// TIA Portal project "topgun_plc" (V16)

(* hardware
DEVICE "S7-1200 station_1"  S7-1200 Station
   slot 0: "Rack_0"  S7-1200 Rack  Rack  V1.0
   slot 1: "PLC_CU"  CPU 1214C DC/DC/DC  6ES7 214-1AG40-0XB0  V4.4
   slot 2: "DI 16/DQ 16x24VDC_1"  6ES7 223-1BL32-0XB0  V2.0
   slot 3: "CB 1241 (RS485)"  CB 1241 (RS485)  6ES7 241-1CH30-1XB0  V1.0
DEVICE "S7-1200 station_2"  S7-1200 Station
   slot 0: "Rack_0"  S7-1200 Rack  Rack  V1.0
   slot 1: "PLC_CAM"  CPU 1214C DC/DC/DC  6ES7 214-1AG40-0XB0  V4.4
*)

// ===== PLC "PLC_CU"  CPU 1214C DC/DC/DC =====

VAR_GLOBAL   // PLC tag table "Default tag table"
   "System_Byte" AT %MB1 : Byte;
   "FirstScan" AT %M1.0 : Bool;
   "DiagStatusUpdate" AT %M1.1 : Bool;
   "AlwaysTRUE" AT %M1.2 : Bool;
   "AlwaysFALSE" AT %M1.3 : Bool;
   "Clock_Byte" AT %MB0 : Byte;
   "Clock_10Hz" AT %M0.0 : Bool;
   "Clock_5Hz" AT %M0.1 : Bool;
   "Clock_2.5Hz" AT %M0.2 : Bool;
   "Clock_2Hz" AT %M0.3 : Bool;
   "Clock_1.25Hz" AT %M0.4 : Bool;
   "Clock_1Hz" AT %M0.5 : Bool;
   "Clock_0.625Hz" AT %M0.6 : Bool;
   "Clock_0.5Hz" AT %M0.7 : Bool;
   "Tag_1" AT %I0.0 : Bool;
   "Tag_2" AT %I0.1 : Bool;
   "Tag_3" AT %I0.2 : Bool;
   "Tag_4" AT %I0.3 : Bool;
   "Tag_5" AT %I2.2 : Bool;
   "Tag_6" AT %I2.3 : Bool;
   "Tag_7" AT %I2.6 : Bool;
   "Tag_8" AT %I2.7 : Bool;
   "Tag_9" AT %ID1000 : DWord;
   "Tag_10" AT %ID1004 : DWord;
   "Tag_11" AT %ID1002 : DWord;
   "Tag_12" AT %ID1006 : DWord;
   "Tag_13" AT %M100.0 : Bool;
   "Tag_14" AT %M100.1 : Bool;
END_VAR

DATA_BLOCK "MB_CONFIG"   // DB2
{ S7_Optimized_Access := 'TRUE' }
VERSION : 0.1
   VAR
      MB_stat : Word;
      MB1_stat : Word;
      MB : TCON_IP_v4;
      MB1 : TCON_IP_v4;
   END_VAR
BEGIN
   MB.RemoteAddress.ADDR[1] := 16#C0;
   MB.RemoteAddress.ADDR[2] := 16#A8;
   MB.RemoteAddress.ADDR[4] := 16#49;
   MB.LocalPort := 502;
   MB1.RemoteAddress.ADDR[1] := 16#C0;
   MB1.RemoteAddress.ADDR[2] := 16#A8;
   MB1.RemoteAddress.ADDR[4] := 16#47;
   MB1.LocalPort := 503;
   MB.InterfaceId := 64;
   MB.ID := 2;
   MB1.InterfaceId := 64;
   MB1.ID := 3;
END_DATA_BLOCK

DATA_BLOCK "MB_DATA"   // DB3
{ S7_Optimized_Access := 'FALSE' }
VERSION : 0.1
   VAR
      DATA : Array[0..64] of Int;
   END_VAR
BEGIN
   DATA[4] := 6;
END_DATA_BLOCK

DATA_BLOCK "Retain_mem"   // DB7
{ S7_Optimized_Access := 'TRUE' }
VERSION : 0.1
   VAR
      Value_HSC1_Save : DWord;
   END_VAR
   VAR RETAIN
      Value_HSC1_Load : DWord;
   END_VAR
   VAR
      Value_HSC2_Save : DWord;
   END_VAR
   VAR RETAIN
      Value_HSC2_Load : DWord;
   END_VAR
   VAR
      Value_Angle1 : Real;
      Value_Angle2 : Real;
      temp1 : Real;
      temp2 : Real;
   END_VAR
BEGIN
END_DATA_BLOCK

ORGANIZATION_BLOCK "Main"   // OB1, LAD, ProgramCycle
TITLE = "Main Program Sweep (Cycle)"
{ S7_Optimized_Access := 'TRUE' }
VERSION : 0.1
   VAR_INPUT
      Initial_Call : Bool;   // Initial call of this OB
      Remanence : Bool;   // =True, if remanent data are available
   END_VAR
BEGIN

REGION Network 1
   // modbus 485
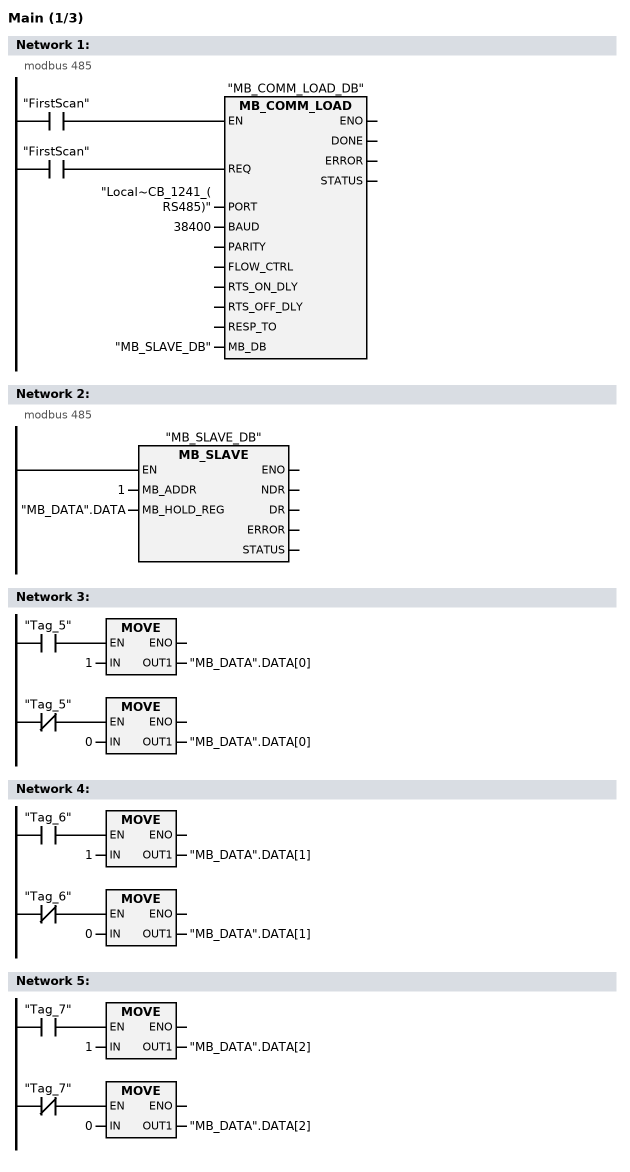
   IF "FirstScan" THEN
       "MB_COMM_LOAD_DB"(REQ := "FirstScan", PORT := "Local~CB_1241_(RS485)", BAUD := 38400, MB_DB := "MB_SLAVE_DB");   // MB_COMM_LOAD
   END_IF;
END_REGION

REGION Network 2
   // modbus 485
   "MB_SLAVE_DB"(MB_ADDR := 1, MB_HOLD_REG := "MB_DATA".DATA);   // MB_SLAVE
END_REGION

REGION Network 3
   RUNG wire#powerrail
      Contact( "Tag_5" )
      Move(in := 1, out1 => "MB_DATA".DATA[0])
   END_RUNG
   RUNG wire#powerrail
      I_Contact( "Tag_5" )
      Move(in := 0, out1 => "MB_DATA".DATA[0])
   END_RUNG
   // the same network as SCL:
   IF "Tag_5" THEN "MB_DATA".DATA[0] := 1; END_IF;
   IF NOT "Tag_5" THEN "MB_DATA".DATA[0] := 0; END_IF;
END_REGION

REGION Network 4
   RUNG wire#powerrail
      Contact( "Tag_6" )
      Move(in := 1, out1 => "MB_DATA".DATA[1])
   END_RUNG
   RUNG wire#powerrail
      I_Contact( "Tag_6" )
      Move(in := 0, out1 => "MB_DATA".DATA[1])
   END_RUNG
   // the same network as SCL:
   IF "Tag_6" THEN "MB_DATA".DATA[1] := 1; END_IF;
   IF NOT "Tag_6" THEN "MB_DATA".DATA[1] := 0; END_IF;
END_REGION

REGION Network 5
   RUNG wire#powerrail
      Contact( "Tag_7" )
      Move(in := 1, out1 => "MB_DATA".DATA[2])
   END_RUNG
   RUNG wire#powerrail
      I_Contact( "Tag_7" )
      Move(in := 0, out1 => "MB_DATA".DATA[2])
   END_RUNG
   // the same network as SCL:
   IF "Tag_7" THEN "MB_DATA".DATA[2] := 1; END_IF;
   IF NOT "Tag_7" THEN "MB_DATA".DATA[2] := 0; END_IF;
END_REGION

REGION Network 6
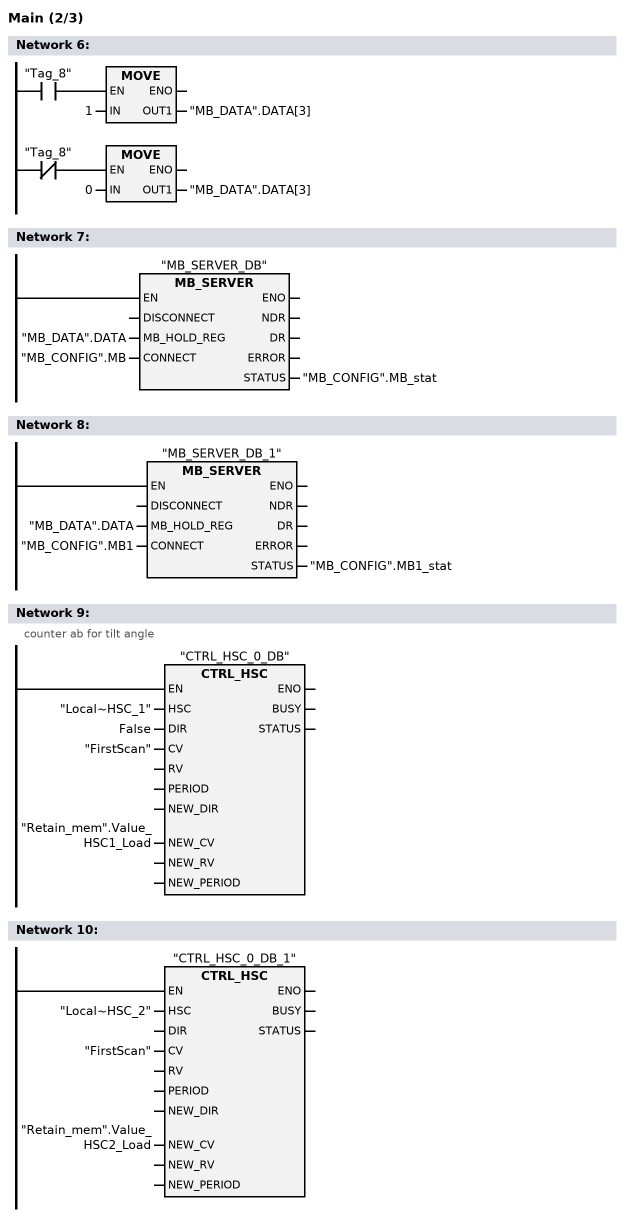
   RUNG wire#powerrail
      Contact( "Tag_8" )
      Move(in := 1, out1 => "MB_DATA".DATA[3])
   END_RUNG
   RUNG wire#powerrail
      I_Contact( "Tag_8" )
      Move(in := 0, out1 => "MB_DATA".DATA[3])
   END_RUNG
   // the same network as SCL:
   IF "Tag_8" THEN "MB_DATA".DATA[3] := 1; END_IF;
   IF NOT "Tag_8" THEN "MB_DATA".DATA[3] := 0; END_IF;
END_REGION

REGION Network 7
   "MB_SERVER_DB"(MB_HOLD_REG := "MB_DATA".DATA, CONNECT := "MB_CONFIG".MB, STATUS => "MB_CONFIG".MB_stat);   // MB_SERVER
END_REGION

REGION Network 8
   "MB_SERVER_DB_1"(MB_HOLD_REG := "MB_DATA".DATA, CONNECT := "MB_CONFIG".MB1, STATUS => "MB_CONFIG".MB1_stat);   // MB_SERVER
END_REGION

REGION Network 9
   // counter ab for tilt angle
   "CTRL_HSC_0_DB"(HSC := "Local~HSC_1",   // CTRL_HSC
                   DIR := False,
                   CV := "FirstScan",
                   NEW_CV := "Retain_mem".Value_HSC1_Load);
END_REGION

REGION Network 10
   "CTRL_HSC_0_DB_1"(HSC := "Local~HSC_2", CV := "FirstScan", NEW_CV := "Retain_mem".Value_HSC2_Load);   // CTRL_HSC
END_REGION

REGION Network 11
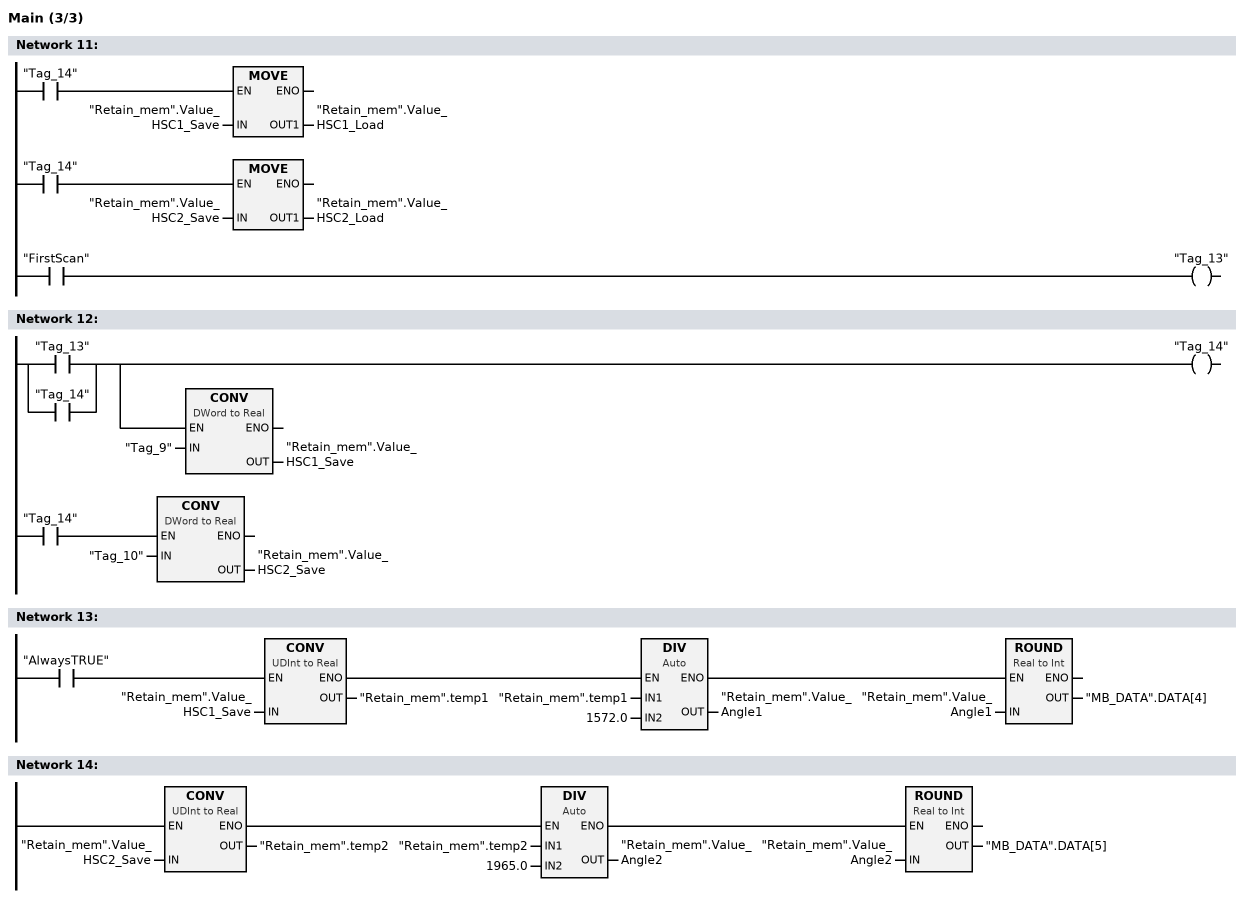
   RUNG wire#powerrail
      Contact( "Tag_14" )
      { S7_GenerateENO := "TRUE" } Move(in := "Retain_mem".Value_HSC1_Save, out1 => "Retain_mem".Value_HSC1_Load)
   END_RUNG
   RUNG wire#powerrail
      Contact( "Tag_14" )
      { S7_GenerateENO := "TRUE" } Move(in := "Retain_mem".Value_HSC2_Save, out1 => "Retain_mem".Value_HSC2_Load)
   END_RUNG
   RUNG wire#powerrail
      Contact( "FirstScan" )
      Coil( "Tag_13" )
   END_RUNG
   // the same network as SCL:
   IF "Tag_14" THEN
       "Retain_mem".Value_HSC1_Load := "Retain_mem".Value_HSC1_Save;
       "Retain_mem".Value_HSC2_Load := "Retain_mem".Value_HSC2_Save;
   END_IF;
   "Tag_13" := "FirstScan";
END_REGION

REGION Network 12
   RUNG wire#powerrail
      Contact( "Tag_13" )
      wire#w1
      Coil( "Tag_14" )
   END_RUNG
   RUNG wire#powerrail
      Contact( "Tag_14" )
   END_RUNG wire#w1
   RUNG wire#w1
      { S7_Templates := "[SrcType := DWord, DestType := Real]" } Convert(in := "Tag_9", out => "Retain_mem".Value_HSC1_Save)
   END_RUNG
   RUNG wire#powerrail
      Contact( "Tag_14" )
      { S7_Templates := "[SrcType := DWord, DestType := Real]" } Convert(in := "Tag_10", out => "Retain_mem".Value_HSC2_Save)
   END_RUNG
   // the same network as SCL:
   "Tag_14" := "Tag_13" OR "Tag_14";
   IF "Tag_14" THEN
       "Retain_mem".Value_HSC1_Save := DWORD_TO_REAL("Tag_9");
       "Retain_mem".Value_HSC2_Save := DWORD_TO_REAL("Tag_10");
   END_IF;
END_REGION

REGION Network 13
   RUNG wire#powerrail
      Contact( "AlwaysTRUE" )
      { S7_Templates := "[SrcType := UDInt, DestType := Real]" } Convert(in := "Retain_mem".Value_HSC1_Save, out => "Retain_mem".temp1)
      Div(in1 := "Retain_mem".temp1, in2 := 1572.0, out => "Retain_mem".Value_Angle1)
      { S7_Templates := "[SrcType := Real, DestType := Int]" } Round(in := "Retain_mem".Value_Angle1, out => "MB_DATA".DATA[4])
   END_RUNG
   // the same network as SCL:
   IF "AlwaysTRUE" THEN
       "Retain_mem".temp1 := UDINT_TO_REAL("Retain_mem".Value_HSC1_Save);
       "Retain_mem".Value_Angle1 := "Retain_mem".temp1 / 1572.0;
       "MB_DATA".DATA[4] := ROUND("Retain_mem".Value_Angle1);
   END_IF;
END_REGION

REGION Network 14
   RUNG wire#powerrail
      { S7_Templates := "[SrcType := UDInt, DestType := Real]" } Convert(in := "Retain_mem".Value_HSC2_Save, out => "Retain_mem".temp2)
      Div(in1 := "Retain_mem".temp2, in2 := 1965.0, out => "Retain_mem".Value_Angle2)
      { S7_Templates := "[SrcType := Real, DestType := Int]" } Round(in := "Retain_mem".Value_Angle2, out => "MB_DATA".DATA[5])
   END_RUNG
   // the same network as SCL:
   "Retain_mem".temp2 := UDINT_TO_REAL("Retain_mem".Value_HSC2_Save);
   "Retain_mem".Value_Angle2 := "Retain_mem".temp2 / 1965.0;
   "MB_DATA".DATA[5] := ROUND("Retain_mem".Value_Angle2);
END_REGION
END_ORGANIZATION_BLOCK

// ===== PLC "PLC_CAM"  CPU 1214C DC/DC/DC =====

DATA_BLOCK "MB_CONFIG"   // DB2
{ S7_Optimized_Access := 'TRUE' }
VERSION : 0.1
   VAR
      MB_stat : Word;
      MB1_stat : Word;
      MB : TCON_IP_v4;
      MB1 : TCON_IP_v4;
   END_VAR
BEGIN
   MB.RemoteAddress.ADDR[1] := 16#C0;
   MB.RemoteAddress.ADDR[2] := 16#A8;
   MB.RemoteAddress.ADDR[4] := 16#49;
   MB.LocalPort := 502;
   MB1.RemoteAddress.ADDR[1] := 16#C0;
   MB1.RemoteAddress.ADDR[2] := 16#A8;
   MB1.RemoteAddress.ADDR[4] := 16#47;
   MB1.LocalPort := 503;
   MB.InterfaceId := 64;
   MB.ID := 2;
   MB1.InterfaceId := 64;
   MB1.ID := 3;
END_DATA_BLOCK

DATA_BLOCK "MB_DATA"   // DB3
{ S7_Optimized_Access := 'FALSE' }
VERSION : 0.1
   VAR
      DATA : Array[0..64] of Int;
   END_VAR
BEGIN
   DATA[4] := 6;
END_DATA_BLOCK

ORGANIZATION_BLOCK "Main"   // OB1, LAD, ProgramCycle
TITLE = "Main Program Sweep (Cycle)"
{ S7_Optimized_Access := 'TRUE' }
VERSION : 0.1
   VAR_INPUT
      Initial_Call : Bool;   // Initial call of this OB
      Remanence : Bool;   // =True, if remanent data are available
   END_VAR
BEGIN

REGION Network 1
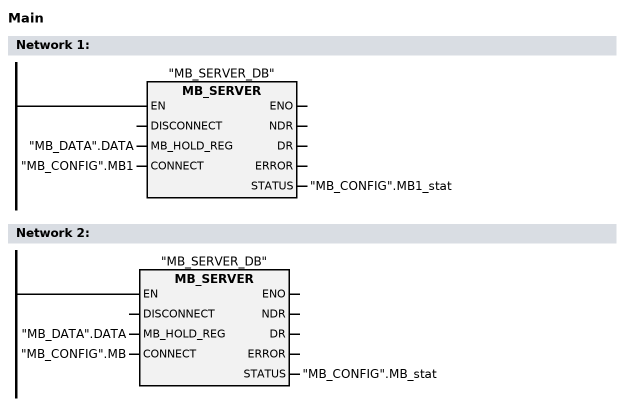
   "MB_SERVER_DB"(MB_HOLD_REG := "MB_DATA".DATA, CONNECT := "MB_CONFIG".MB1, STATUS => "MB_CONFIG".MB1_stat);   // MB_SERVER
END_REGION

REGION Network 2
   "MB_SERVER_DB"(MB_HOLD_REG := "MB_DATA".DATA, CONNECT := "MB_CONFIG".MB, STATUS => "MB_CONFIG".MB_stat);   // MB_SERVER
END_REGION
END_ORGANIZATION_BLOCK